// TwinCAT 3 PLC project CallingStandardFunction
// ProgramVersion: 3.1.4023.0
// libraries:
//   Tc2_Standard, * (Beckhoff Automation GmbH)
//   Tc2_System, * (Beckhoff Automation GmbH)
//   Tc3_Module, * (Beckhoff Automation GmbH)
// project tree:
//   / PlcTask.TcTTO
//   POUs/ Call_Std_Func.TcPOU, MAIN.TcPOU (not stored)

CONFIGURATION CallingStandardFunction
    RESOURCE PLC ON TwinCAT3
        TASK PlcTask(INTERVAL := T#10ms, PRIORITY := 20);
        PROGRAM MAIN WITH PlcTask : MAIN;
    END_RESOURCE
END_CONFIGURATION

// ---- POUs/Call_Std_Func.TcPOU
PROGRAM Call_Std_Func
VAR
	Start: BOOL;
	Stop: BOOL;
	Motor1: BOOL;
	Motor2: BOOL;
	Timer1: TON;
	Done: BOOL;
	ElapsedTime: TIME;
	Timer2: TON;
END_VAR

IF Start THEN
	Motor1 := TRUE;
END_IF

IF Motor1 THEN
	Timer1(IN:=TRUE , PT:= T#5S, Q=>Done , ET=> ElapsedTime);
END_IF

IF TIMER1.Q THEN
	Timer1(IN := FALSE);
	Motor2 := TRUE;
END_IF

IF Stop THEN
	Motor1 := FALSE;
	Motor2 := FALSE;
END_IF

END_PROGRAM
